PROGRAM MAIN
VAR
END_VAR

END_PROGRAM

(* stored: Version 1.1.0.1
   POU MAIN: Id {99702faa-dee6-4436-b0d6-1042ea702d18} *)
